{region '#Template'}
	{attribute 'Version' := '1.0.0.0'}
	{attribute 'Tags' := '"LCID": "1031", "Text": "AC, Aggregates, ERC, Plate"'}
	{attribute 'Tags' := '"LCID": "1033", "Text": "AC, Aggregates, ERC, Plate"'}
	{attribute 'Description' := '"LCID": "1031", "Text": "Aggregat Energie Rückgewinnung Platte mit Bypass"'}
	{attribute 'Description' := '"LCID": "1033", "Text": "Aggregate energy recovery plate with bypass"'}
{endregion}
FUNCTION_BLOCK FB_BA_AC_ErcPl_02 EXTENDS FB_BA_AggregateB
VAR_INPUT
	fSpTSuA					: REAL;
	fTSuA					: REAL;
	bDehumf					: BOOL;
	fTExhA					: REAL;
	fTExtA					: REAL;
	fTWth					: REAL;
END_VAR
VAR_OUTPUT
	fPresentValue			: REAL;				
	eAction					: E_BA_Action;
	bActiveSeqCtrl			: BOOL;	
END_VAR
VAR_INPUT CONSTANT
	TSuACtrl				: FB_BA_AC_ErcTSuACtrl;								 
	TExhACtrl				: FB_BA_PID_Sp;														
	DiffPrssSwi				: FB_BA_SensorBinary_IO;							
	IcePrtcRamp				: FB_BA_RampLimitIncrease;								
	Dmp						: FB_BA_ActuatorAnalog;
	ByDmp					: FB_BA_ActuatorAnalog;					
END_VAR
VAR
	Inv						: FB_BA_Chrct02;	
END_VAR
VAR // added by the converter: edge detectors and wires of the graphical bodies
    _w1 : ANY;
END_VAR

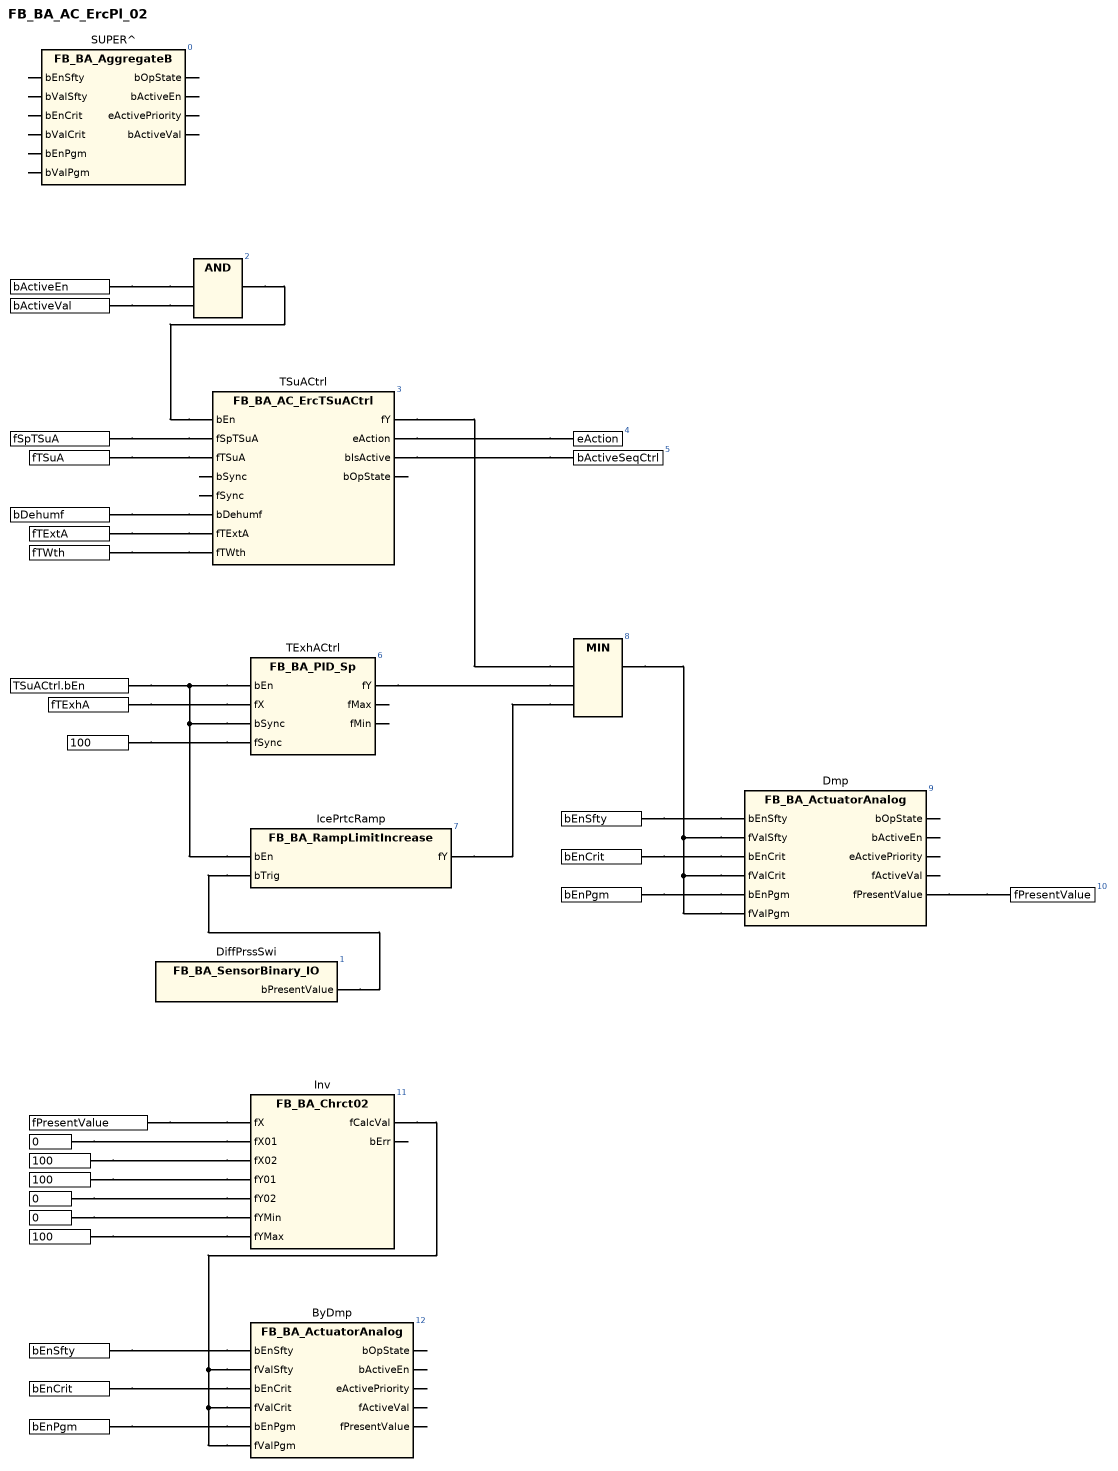
SUPER^(); // FB_BA_AggregateB
DiffPrssSwi(); // FB_BA_SensorBinary_IO
TSuACtrl(
    bEn := bActiveEn AND bActiveVal,
    fSpTSuA := fSpTSuA,
    fTSuA := fTSuA,
    bDehumf := bDehumf,
    fTExtA := fTExtA,
    fTWth := fTWth); // FB_BA_AC_ErcTSuACtrl
eAction := TSuACtrl.eAction;
bActiveSeqCtrl := TSuACtrl.bIsActive;
TExhACtrl(bEn := TSuACtrl.bEn, fX := fTExhA, bSync := TSuACtrl.bEn, fSync := 100); // FB_BA_PID_Sp
IcePrtcRamp(bEn := TSuACtrl.bEn, bTrig := DiffPrssSwi.bPresentValue); // FB_BA_RampLimitIncrease
_w1 := MIN(TSuACtrl.fY, TExhACtrl.fY, IcePrtcRamp.fY);
Dmp(
    bEnSfty := bEnSfty,
    fValSfty := _w1,
    bEnCrit := bEnCrit,
    fValCrit := _w1,
    bEnPgm := bEnPgm,
    fValPgm := _w1); // FB_BA_ActuatorAnalog
fPresentValue := Dmp.fPresentValue;
Inv(fX := fPresentValue, fX01 := 0, fX02 := 100, fY01 := 100, fY02 := 0, fYMin := 0, fYMax := 100); // FB_BA_Chrct02
ByDmp(
    bEnSfty := bEnSfty,
    fValSfty := Inv.fCalcVal,
    bEnCrit := bEnCrit,
    fValCrit := Inv.fCalcVal,
    bEnPgm := bEnPgm,
    fValPgm := Inv.fCalcVal); // FB_BA_ActuatorAnalog

METHOD FB_init : BOOL
VAR_INPUT
	bInitRetains : BOOL; // if TRUE, the retain variables are initialized (warm start / cold start)
	bInCopyCode : BOOL;  // if TRUE, the instance afterwards gets moved into the copy code (online change)
END_VAR
TSuACtrl.iParent									:= THIS^;	
TSuACtrl.iLabel										:= LblCmpAC.ERC_TSuACtrl;
TSuACtrl.sObjectName								:= '{Idx=21}';										 
TSuACtrl.eDPADMode									:= E_BA_DPADMode.eInclude;								

TExhACtrl.iParent									:= THIS^;	
TExhACtrl.iLabel									:= LblCmpAC.ERC_TExhACtrl;
TExhACtrl.sObjectName								:= '{Idx=22}';										 
TExhACtrl.eDPADMode									:= E_BA_DPADMode.eInclude;
TExhACtrl.Sp.fValueRm 								:= 6.0;
TExhACtrl.Ctrl.eActionRm							:= E_BA_Action.eDirect;

DiffPrssSwi.iParent									:= THIS^;
DiffPrssSwi.iLabel									:= LblCmpAC.ERC_DiffPrssSwi;												 										 
DiffPrssSwi.sObjectName								:= '{Idx=21}';
DiffPrssSwi.eDPADMode								:= E_BA_DPADMode.eInclude;
DiffPrssSwi.Input.iLabel							:= LblFunctions_OperationalMessage;	
DiffPrssSwi.Input.sObjectName						:= '{Idx=01}';	
DiffPrssSwi.Input.ePolarity							:= E_BA_Polarity.eReverse;
DiffPrssSwi.Input.sActiveText 						:= txtEvent_Triggered;
DiffPrssSwi.Input.sInactiveText 					:= txtEvent_Normal;
DiffPrssSwi.Input.nEventClassID						:= EventClasses.AlarmTechnicalExtended;
DiffPrssSwi.Input.aEventTransitionText[1]			:= txtEvent_Triggered;
DiffPrssSwi.Input.aEventTransitionText[2]			:= txtEvent_Error;
DiffPrssSwi.Input.aEventTransitionText[3]			:= txtEvent_Normal;
DiffPrssSwi.Input.bEventDetectionEnable				:= TRUE;
DiffPrssSwi.Input.eEnPlantLock						:= E_BA_LockPriority.eNoLock;	


IcePrtcRamp.iParent									:= THIS^;	
IcePrtcRamp.iLabel									:= LblCmpAC.ERC_IcePrtcRamp;
IcePrtcRamp.sObjectName								:= '{Idx=21}';										 
IcePrtcRamp.eDPADMode								:= E_BA_DPADMode.eIncludeDescription;
IcePrtcRamp.TiUp.fValueRm							:= 1200;

Dmp.iParent											:= THIS^;
Dmp.iLabel											:= LblCmpAC.ERC_Dmp;	
Dmp.sObjectName										:= '{Idx=21}';										 
Dmp.eDPADMode										:= E_BA_DPADMode.eInclude;
Dmp.Mdlt.fResolution 								:= 0.003814755;
Dmp.Mdlt.fScaleOffset 								:= 0;

ByDmp.iParent										:= THIS^;
ByDmp.iLabel										:= LblCmpAC.ERC_ByDmp;	
ByDmp.sObjectName									:= '{Idx=22}';										 
ByDmp.eDPADMode										:= E_BA_DPADMode.eInclude;
ByDmp.Mdlt.fResolution 								:= 0.003814755;
ByDmp.Mdlt.fScaleOffset 							:= 0;
END_METHOD

END_FUNCTION_BLOCK

(* stored: Version 1.1.0.1, ProductVersion 3.1.4024.9
   POU FB_BA_AC_ErcPl_02: Id {a40c3197-7d5d-406c-bfa7-c0810e8d4c90}, SpecialFunc None
   Method FB_init: Id {443efafb-1b45-48fb-ac7d-5e0cab38e44a} *)
